LIN {X 0,Y 73.676,Z 293.865,A -85,B 0,C 180,E1 -30414.523,E2 -30414.523} C_VEL
LIN {X 0,Y 74.432,Z 292.814,A -85,B 0,C 180,E1 -30419.997,E2 -30419.997} C_VEL
LIN {X 0,Y 73.431,Z 293.677,A -85,B 0,C 180,E1 -30426.603,E2 -30426.603} C_VEL
LIN {X 0,Y 72.907,Z 294.465,A -85,B 0,C 180,E1 -30431.113,E2 -30431.113} C_VEL
LIN {X 0,Y 72.2,Z 295.883,A -85,B 0,C 180,E1 -30436.976,E2 -30436.976} C_VEL
LIN {X 0,Y 70.658,Z 298.436,A -85,B 0,C 180,E1 -30443.441,E2 -30443.441} C_VEL
LIN {X 0,Y 69.644,Z 299.949,A -85,B 0,C 180,E1 -30447.198,E2 -30447.198} C_VEL
LIN {X 0,Y 67.365,Z 302.892,A -85,B 0,C 180,E1 -30453.425,E2 -30453.425} C_VEL
LIN {X 0,Y 63.424,Z 307.476,A -85,B 0,C 180,E1 -30464.197,E2 -30464.197} C_VEL
LIN {X 0,Y 61.844,Z 310.777,A -85,B 0,C 180,E1 -30475.376,E2 -30475.376} C_VEL
LIN {X 0,Y 62.437,Z 312.643,A -85,B 0,C 180,E1 -30484.215,E2 -30484.215} C_VEL
LIN {X 0,Y 67.085,Z 314.547,A -85,B 0,C 180,E1 -30497.906,E2 -30497.906} C_VEL
LIN {X 0,Y 71.285,Z 314.971,A -85,B 0,C 180,E1 -30504.342,E2 -30504.342} C_VEL
LIN {X 0,Y 76.406,Z 314.961,A -85,B 0,C 180,E1 -30510,E2 -30510} C_VEL
LIN {X 0,Y 70.707,Z 314.927,A -85,B 0,C 180,E1 -30516.332,E2 -30516.332} C_VEL
LIN {X 0,Y 65.554,Z 314.211,A -85,B 0,C 180,E1 -30525.243,E2 -30525.243} C_VEL
LIN {X 0,Y 62.272,Z 312.421,A -85,B 0,C 180,E1 -30536.836,E2 -30536.836} C_VEL
LIN {X 0,Y 61.936,Z 310.037,A -85,B 0,C 180,E1 -30547.417,E2 -30547.417} C_VEL
LIN {X 0,Y 64.396,Z 306.165,A -85,B 0,C 180,E1 -30559.098,E2 -30559.098} C_VEL
LIN {X 0,Y 67.359,Z 302.893,A -85,B 0,C 180,E1 -30566.583,E2 -30566.583} C_VEL
LIN {X 0,Y 69.605,Z 299.971,A -85,B 0,C 180,E1 -30572.791,E2 -30572.791} C_VEL
LIN {X 0,Y 71.492,Z 297.039,A -85,B 0,C 180,E1 -30579.878,E2 -30579.878} C_VEL
LIN {X 0,Y 72.19,Z 295.89,A -85,B 0,C 180,E1 -30583.022,E2 -30583.022} C_VEL
LIN {X 0,Y 72.906,Z 294.466,A -85,B 0,C 180,E1 -30588.887,E2 -30588.887} C_VEL
LIN {X 0,Y 73.634,Z 293.478,A -85,B 0,C 180,E1 -30594.526,E2 -30594.526} C_VEL
LIN {X 0,Y 74.44,Z 292.808,A -85,B 0,C 180,E1 -30600.003,E2 -30600.003} C_VEL
LIN {X 0,Y 73.487,Z 294.094,A -85,B 0,C 180,E1 -30606.279,E2 -30606.279} C_VEL
LIN {X 0,Y 72.295,Z 295.22,A -85,B 0,C 180,E1 -30608.406,E2 -30608.406} C_VEL
LIN {X 0,Y 69.831,Z 297.145,A -85,B 0,C 180,E1 -30610.311,E2 -30610.311} C_VEL
LIN {X 0,Y 67.327,Z 298.912,A -85,B 0,C 180,E1 -30611.434,E2 -30611.434} C_VEL
LIN {X 0,Y 57.475,Z 304.685,A -85,B 0,C 180,E1 -30614.417,E2 -30614.417} C_VEL
LIN {X 0,Y 48.227,Z 309.171,A -85,B 0,C 180,E1 -30618.7,E2 -30618.7} C_VEL
LIN {X 0,Y 38.879,Z 312.786,A -85,B 0,C 180,E1 -30625.335,E2 -30625.335} C_VEL
LIN {X 0,Y 33.035,Z 314.591,A -85,B 0,C 180,E1 -30631.685,E2 -30631.685} C_VEL
LIN {X 0,Y 23.562,Z 317.062,A -85,B 0,C 180,E1 -30653.377,E2 -30653.377} C_VEL
LIN {X 0,Y 20.768,Z 317.664,A -85,B 0,C 180,E1 -30670.221,E2 -30670.221} C_VEL
LIN {X 0,Y 20.025,Z 317.831,A -85,B 0,C 180,E1 -30690,E2 -30690} C_VEL
LIN {X 0,Y 20.768,Z 317.664,A -85,B 0,C 180,E1 -30709.779,E2 -30709.779} C_VEL
LIN {X 0,Y 23.562,Z 317.062,A -85,B 0,C 180,E1 -30726.623,E2 -30726.623} C_VEL
LIN {X 0,Y 33.035,Z 314.591,A -85,B 0,C 180,E1 -30748.315,E2 -30748.315} C_VEL
LIN {X 0,Y 41.94,Z 311.634,A -85,B 0,C 180,E1 -30757.168,E2 -30757.168} C_VEL
LIN {X 0,Y 51.467,Z 307.64,A -85,B 0,C 180,E1 -30762.914,E2 -30762.914} C_VEL
LIN {X 0,Y 61.31,Z 302.505,A -85,B 0,C 180,E1 -30766.98,E2 -30766.98} C_VEL
LIN {X 0,Y 64.639,Z 300.584,A -85,B 0,C 180,E1 -30768.106,E2 -30768.106} C_VEL
LIN {X 0,Y 66.852,Z 298.764,A -85,B 0,C 180,E1 -30771.244,E2 -30771.244} C_VEL
LIN {X 0,Y 67.395,Z 298.046,A -85,B 0,C 180,E1 -30774.011,E2 -30774.011} C_VEL
LIN {X 0,Y 68.442,Z 296.911,A -85,B 0,C 180,E1 -30779.997,E2 -30779.997} C_VEL
LIN {X 0,Y 67.508,Z 297.553,A -85,B 0,C 180,E1 -30785.972,E2 -30785.972} C_VEL
LIN {X 0,Y 66.682,Z 298.624,A -85,B 0,C 180,E1 -30792.165,E2 -30792.165} C_VEL
LIN {X 0,Y 65.976,Z 299.629,A -85,B 0,C 180,E1 -30796.524,E2 -30796.524} C_VEL
LIN {X 0,Y 64.231,Z 301.578,A -85,B 0,C 180,E1 -30802.513,E2 -30802.513} C_VEL
LIN {X 0,Y 62.878,Z 303.159,A -85,B 0,C 180,E1 -30806.6,E2 -30806.6} C_VEL
LIN {X 0,Y 61.26,Z 304.717,A -85,B 0,C 180,E1 -30810.636,E2 -30810.636} C_VEL
LIN {X 0,Y 58.689,Z 307.105,A -85,B 0,C 180,E1 -30816.776,E2 -30816.776} C_VEL
LIN {X 0,Y 55.19,Z 311.025,A -85,B 0,C 180,E1 -30830.454,E2 -30830.454} C_VEL
LIN {X 0,Y 55.208,Z 313.32,A -85,B 0,C 180,E1 -30843.003,E2 -30843.003} C_VEL
LIN {X 0,Y 58.568,Z 314.807,A -85,B 0,C 180,E1 -30856.114,E2 -30856.114} C_VEL
LIN {X 0,Y 63.482,Z 315.319,A -85,B 0,C 180,E1 -30865.075,E2 -30865.075} C_VEL
LIN {X 0,Y 67.402,Z 315.229,A -85,B 0,C 180,E1 -30870,E2 -30870} C_VEL
LIN {X 0,Y 62.433,Z 315.236,A -85,B 0,C 180,E1 -30876.463,E2 -30876.463} C_VEL
LIN {X 0,Y 58.179,Z 314.746,A -85,B 0,C 180,E1 -30884.909,E2 -30884.909} C_VEL
LIN {X 0,Y 54.905,Z 312.671,A -85,B 0,C 180,E1 -30900.797,E2 -30900.797} C_VEL
LIN {X 0,Y 55.809,Z 309.953,A -85,B 0,C 180,E1 -30913.831,E2 -30913.831} C_VEL
LIN {X 0,Y 59.644,Z 306.186,A -85,B 0,C 180,E1 -30925.57,E2 -30925.57} C_VEL
LIN {X 0,Y 61.252,Z 304.718,A -85,B 0,C 180,E1 -30929.376,E2 -30929.376} C_VEL
LIN {X 0,Y 62.893,Z 303.139,A -85,B 0,C 180,E1 -30933.454,E2 -30933.454} C_VEL
LIN {X 0,Y 64.239,Z 301.573,A -85,B 0,C 180,E1 -30937.489,E2 -30937.489} C_VEL
LIN {X 0,Y 65.956,Z 299.631,A -85,B 0,C 180,E1 -30943.534,E2 -30943.534} C_VEL
LIN {X 0,Y 66.682,Z 298.625,A -85,B 0,C 180,E1 -30947.835,E2 -30947.835} C_VEL
LIN {X 0,Y 67.507,Z 297.554,A -85,B 0,C 180,E1 -30954.028,E2 -30954.028} C_VEL
LIN {X 0,Y 68.451,Z 296.906,A -85,B 0,C 180,E1 -30960.003,E2 -30960.003} C_VEL
LIN {X 0,Y 67.396,Z 298.046,A -85,B 0,C 180,E1 -30965.989,E2 -30965.989} C_VEL
LIN {X 0,Y 66.842,Z 298.771,A -85,B 0,C 180,E1 -30968.756,E2 -30968.756} C_VEL
LIN {X 0,Y 64.638,Z 300.584,A -85,B 0,C 180,E1 -30971.891,E2 -30971.891} C_VEL
LIN {X 0,Y 57.475,Z 304.685,A -85,B 0,C 180,E1 -30974.417,E2 -30974.417} C_VEL
LIN {X 0,Y 52.268,Z 307.16,A -85,B 0,C 180,E1 -30975.88,E2 -30975.88} C_VEL
LIN {X 0,Y 46.76,Z 309.424,A -85,B 0,C 180,E1 -30976.537,E2 -30976.537} C_VEL
LIN {X 0,Y 35.413,Z 312.966,A -85,B 0,C 180,E1 -30977.654,E2 -30977.654} C_VEL
LIN {X 0,Y 28.967,Z 314.652,A -85,B 0,C 180,E1 -30980.959,E2 -30980.959} C_VEL
LIN {X 0,Y 28.103,Z 314.782,A -85,B 0,C 180,E1 -30981.829,E2 -30981.829} C_VEL
LIN {X 0,Y 18.343,Z 316.85,A -85,B 0,C 180,E1 -30999.98,E2 -30999.98} C_VEL
LIN {X 0,Y 14.272,Z 317.452,A -85,B 0,C 180,E1 -31020.499,E2 -31020.499} C_VEL
LIN {X 0,Y 12.932,Z 317.619,A -85,B 0,C 180,E1 -31050,E2 -31050} C_VEL
LIN {X 0,Y 14.272,Z 317.452,A -85,B 0,C 180,E1 -31079.501,E2 -31079.501} C_VEL
LIN {X 0,Y 18.343,Z 316.85,A -85,B 0,C 180,E1 -31100.02,E2 -31100.02} C_VEL
LIN {X 0,Y 29.911,Z 314.379,A -85,B 0,C 180,E1 -31120.026,E2 -31120.026} C_VEL
LIN {X 0,Y 39.721,Z 311.422,A -85,B 0,C 180,E1 -31126.688,E2 -31126.688} C_VEL
LIN {X 0,Y 49.842,Z 307.428,A -85,B 0,C 180,E1 -31130.762,E2 -31130.762} C_VEL
LIN {X 0,Y 60.104,Z 302.292,A -85,B 0,C 180,E1 -31133.638,E2 -31133.638} C_VEL
LIN {X 0,Y 61.567,Z 301.26,A -85,B 0,C 180,E1 -31136.724,E2 -31136.724} C_VEL
LIN {X 0,Y 62.204,Z 300.755,A -85,B 0,C 180,E1 -31139.996,E2 -31139.996} C_VEL
LIN {X 0,Y 61.149,Z 301.337,A -85,B 0,C 180,E1 -31146.596,E2 -31146.596} C_VEL
LIN {X 0,Y 60.018,Z 302.426,A -85,B 0,C 180,E1 -31153.54,E2 -31153.54} C_VEL
LIN {X 0,Y 58.976,Z 303.467,A -85,B 0,C 180,E1 -31157.574,E2 -31157.574} C_VEL
LIN {X 0,Y 57.606,Z 304.623,A -85,B 0,C 180,E1 -31161.465,E2 -31161.465} C_VEL
LIN {X 0,Y 55.306,Z 306.438,A -85,B 0,C 180,E1 -31167.189,E2 -31167.189} C_VEL
LIN {X 0,Y 51.729,Z 309.05,A -85,B 0,C 180,E1 -31175.398,E2 -31175.398} C_VEL
LIN {X 0,Y 48.707,Z 311.604,A -85,B 0,C 180,E1 -31186.169,E2 -31186.169} C_VEL
LIN {X 0,Y 48.237,Z 314.159,A -85,B 0,C 180,E1 -31204.082,E2 -31204.082} C_VEL
LIN {X 0,Y 50.802,Z 315.149,A -85,B 0,C 180,E1 -31215.539,E2 -31215.539} C_VEL
LIN {X 0,Y 56.301,Z 315.561,A -85,B 0,C 180,E1 -31226.933,E2 -31226.933} C_VEL
LIN {X 0,Y 58.456,Z 315.495,A -85,B 0,C 180,E1 -31230,E2 -31230} C_VEL
LIN {X 0,Y 53.713,Z 315.497,A -85,B 0,C 180,E1 -31237.518,E2 -31237.518} C_VEL
LIN {X 0,Y 50.266,Z 315.063,A -85,B 0,C 180,E1 -31246.238,E2 -31246.238} C_VEL
LIN {X 0,Y 48.014,Z 313.88,A -85,B 0,C 180,E1 -31258.579,E2 -31258.579} C_VEL
LIN {X 0,Y 49.072,Z 311.272,A -85,B 0,C 180,E1 -31275.732,E2 -31275.732} C_VEL
LIN {X 0,Y 53.182,Z 308.076,A -85,B 0,C 180,E1 -31288.094,E2 -31288.094} C_VEL
LIN {X 0,Y 55.302,Z 306.438,A -85,B 0,C 180,E1 -31292.82,E2 -31292.82} C_VEL
LIN {X 0,Y 57.608,Z 304.622,A -85,B 0,C 180,E1 -31298.536,E2 -31298.536} C_VEL
LIN {X 0,Y 58.962,Z 303.468,A -85,B 0,C 180,E1 -31302.468,E2 -31302.468} C_VEL
LIN {X 0,Y 60.004,Z 302.434,A -85,B 0,C 180,E1 -31306.456,E2 -31306.456} C_VEL
LIN {X 0,Y 61.148,Z 301.338,A -85,B 0,C 180,E1 -31313.404,E2 -31313.404} C_VEL
LIN {X 0,Y 62.211,Z 300.752,A -85,B 0,C 180,E1 -31320.004,E2 -31320.004} C_VEL
LIN {X 0,Y 61.569,Z 301.259,A -85,B 0,C 180,E1 -31323.275,E2 -31323.275} C_VEL
LIN {X 0,Y 60.103,Z 302.292,A -85,B 0,C 180,E1 -31326.359,E2 -31326.359} C_VEL
LIN {X 0,Y 49.841,Z 307.428,A -85,B 0,C 180,E1 -31329.232,E2 -31329.232} C_VEL
LIN {X 0,Y 39.721,Z 311.422,A -85,B 0,C 180,E1 -31333.311,E2 -31333.311} C_VEL
LIN {X 0,Y 29.911,Z 314.379,A -85,B 0,C 180,E1 -31339.973,E2 -31339.973} C_VEL
LIN {X 0,Y 28.103,Z 314.782,A -85,B 0,C 180,E1 -31341.829,E2 -31341.829} C_VEL
LIN {X 0,Y 22.824,Z 315.916,A -85,B 0,C 180,E1 -31347.349,E2 -31347.349} C_VEL
LIN {X 0,Y 17.343,Z 316.751,A -85,B 0,C 180,E1 -31353.544,E2 -31353.544} C_VEL
LIN {X 0,Y 7.303,Z 317.435,A -85,B 0,C 180,E1 -31387.187,E2 -31387.187} C_VEL
LIN {X 0,Y 7.44,Z 317.287,A -85,B 0,C 180,E1 -31452.841,E2 -31452.841} C_VEL
LIN {X 0,Y 14.811,Z 316.638,A -85,B 0,C 180,E1 -31481.619,E2 -31481.619} C_VEL
LIN {X 0,Y 28.281,Z 314.167,A -85,B 0,C 180,E1 -31493.729,E2 -31493.729} C_VEL
LIN {X 0,Y 38.706,Z 311.21,A -85,B 0,C 180,E1 -31497.009,E2 -31497.009} C_VEL
LIN {X 0,Y 49.203,Z 307.215,A -85,B 0,C 180,E1 -31499.006,E2 -31499.006} C_VEL
LIN {X 0,Y 55.771,Z 304.239,A -85,B 0,C 180,E1 -31499.996,E2 -31499.996} C_VEL
LIN {X 0,Y 54.505,Z 304.848,A -85,B 0,C 180,E1 -31507.404,E2 -31507.404} C_VEL
LIN {X 0,Y 52.596,Z 306.118,A -85,B 0,C 180,E1 -31515.496,E2 -31515.496} C_VEL
LIN {X 0,Y 51.7,Z 306.717,A -85,B 0,C 180,E1 -31517.909,E2 -31517.909} C_VEL
LIN {X 0,Y 49.646,Z 308.09,A -85,B 0,C 180,E1 -31522.669,E2 -31522.669} C_VEL
LIN {X 0,Y 45.47,Z 310.437,A -85,B 0,C 180,E1 -31531.779,E2 -31531.779} C_VEL
LIN {X 0,Y 41.435,Z 313.169,A -85,B 0,C 180,E1 -31547.278,E2 -31547.278} C_VEL
LIN {X 0,Y 42.112,Z 315.318,A -85,B 0,C 180,E1 -31570.502,E2 -31570.502} C_VEL
LIN {X 0,Y 45.091,Z 315.757,A -85,B 0,C 180,E1 -31581.033,E2 -31581.033} C_VEL
LIN {X 0,Y 49.61,Z 315.758,A -85,B 0,C 180,E1 -31590,E2 -31590} C_VEL
LIN {X 0,Y 43.44,Z 315.544,A -85,B 0,C 180,E1 -31603.919,E2 -31603.919} C_VEL
LIN {X 0,Y 40.846,Z 314.409,A -85,B 0,C 180,E1 -31621.076,E2 -31621.076} C_VEL
LIN {X 0,Y 42.402,Z 312.317,A -85,B 0,C 180,E1 -31638.479,E2 -31638.479} C_VEL
LIN {X 0,Y 48.023,Z 308.977,A -85,B 0,C 180,E1 -31653.962,E2 -31653.962} C_VEL
LIN {X 0,Y 49.636,Z 308.095,A -85,B 0,C 180,E1 -31657.32,E2 -31657.32} C_VEL
LIN {X 0,Y 51.695,Z 306.717,A -85,B 0,C 180,E1 -31662.11,E2 -31662.11} C_VEL
LIN {X 0,Y 52.574,Z 306.128,A -85,B 0,C 180,E1 -31664.497,E2 -31664.497} C_VEL
LIN {X 0,Y 54.481,Z 304.859,A -85,B 0,C 180,E1 -31672.592,E2 -31672.592} C_VEL
LIN {X 0,Y 55.769,Z 304.24,A -85,B 0,C 180,E1 -31680.004,E2 -31680.004} C_VEL
LIN {X 0,Y 45.698,Z 308.747,A -85,B 0,C 180,E1 -31681.54,E2 -31681.54} C_VEL
LIN {X 0,Y 35.221,Z 312.362,A -85,B 0,C 180,E1 -31683.89,E2 -31683.89} C_VEL
LIN {X 0,Y 25.513,Z 314.73,A -85,B 0,C 180,E1 -31687.675,E2 -31687.675} C_VEL
LIN {X 0,Y 14.811,Z 316.638,A -85,B 0,C 180,E1 -31698.381,E2 -31698.381} C_VEL
LIN {X 0,Y 8.809,Z 317.24,A -85,B 0,C 180,E1 -31717.08,E2 -31717.08} C_VEL
LIN {X 0,Y 5.826,Z 317.408,A -85,B 0,C 180,E1 -31770,E2 -31770} C_VEL
LIN {X 0,Y 7.44,Z 317.287,A -85,B 0,C 180,E1 -31812.841,E2 -31812.841} C_VEL
LIN {X 0,Y 10.157,Z 317.105,A -85,B 0,C 180,E1 -31831.608,E2 -31831.608} C_VEL
LIN {X 0,Y 16.471,Z 316.308,A -85,B 0,C 180,E1 -31852.457,E2 -31852.457} C_VEL
LIN {X 0,Y 27.155,Z 314.271,A -85,B 0,C 180,E1 -31865.805,E2 -31865.805} C_VEL
LIN {X 0,Y 32.844,Z 312.828,A -85,B 0,C 180,E1 -31867.673,E2 -31867.673} C_VEL
LIN {X 0,Y 34.762,Z 312.328,A -85,B 0,C 180,E1 -31867.704,E2 -31867.704} C_VEL
LIN {X 0,Y 42.531,Z 309.777,A -85,B 0,C 180,E1 -31867.493,E2 -31867.493} C_VEL
LIN {X 0,Y 47.29,Z 308.048,A -85,B 0,C 180,E1 -31868.542,E2 -31868.542} C_VEL
LIN {X 0,Y 44.164,Z 309.551,A -85,B 0,C 180,E1 -31877.296,E2 -31877.296} C_VEL
LIN {X 0,Y 39.45,Z 311.758,A -85,B 0,C 180,E1 -31887.034,E2 -31887.034} C_VEL
LIN {X 0,Y 35.792,Z 313.416,A -85,B 0,C 180,E1 -31898.24,E2 -31898.24} C_VEL
LIN {X 0,Y 34.255,Z 315.569,A -85,B 0,C 180,E1 -31925.775,E2 -31925.775} C_VEL
LIN {X 0,Y 36.636,Z 316.012,A -85,B 0,C 180,E1 -31938.94,E2 -31938.94} C_VEL
LIN {X 0,Y 40.88,Z 316.018,A -85,B 0,C 180,E1 -31950,E2 -31950} C_VEL
LIN {X 0,Y 36.076,Z 315.941,A -85,B 0,C 180,E1 -31963.106,E2 -31963.106} C_VEL
LIN {X 0,Y 33.803,Z 314.999,A -85,B 0,C 180,E1 -31983.744,E2 -31983.744} C_VEL
LIN {X 0,Y 36.495,Z 313.022,A -85,B 0,C 180,E1 -32004.717,E2 -32004.717} C_VEL
LIN {X 0,Y 39.438,Z 311.758,A -85,B 0,C 180,E1 -32013.001,E2 -32013.001} C_VEL
LIN {X 0,Y 44.162,Z 309.551,A -85,B 0,C 180,E1 -32022.713,E2 -32022.713} C_VEL
LIN {X 0,Y 47.271,Z 308.057,A -85,B 0,C 180,E1 -32031.455,E2 -32031.455} C_VEL
LIN {X 0,Y 42.531,Z 309.777,A -85,B 0,C 180,E1 -32032.504,E2 -32032.504} C_VEL
LIN {X 0,Y 35.456,Z 312.15,A -85,B 0,C 180,E1 -32032.336,E2 -32032.336} C_VEL
LIN {X 0,Y 28.399,Z 313.955,A -85,B 0,C 180,E1 -32031.837,E2 -32031.837} C_VEL
LIN {X 0,Y 14.269,Z 316.426,A -85,B 0,C 180,E1 -32030.086,E2 -32030.086} C_VEL
LIN {X 0,Y 7.252,Z 317.029,A -85,B 0,C 180,E1 -32025.719,E2 -32025.719} C_VEL
LIN {X 0,Y 1.286,Z 317.196,A -85,B 0,C 180,E1 -31950,E2 -31950} C_VEL
LIN {X 0,Y 7.252,Z 317.029,A -85,B 0,C 180,E1 -31874.281,E2 -31874.281} C_VEL
LIN {X 0,Y 14.269,Z 316.426,A -85,B 0,C 180,E1 -31869.914,E2 -31869.914} C_VEL
LIN {X 0,Y 28.399,Z 313.955,A -85,B 0,C 180,E1 -31868.163,E2 -31868.163} C_VEL
LIN {X 0,Y 34.762,Z 312.328,A -85,B 0,C 180,E1 -31867.704,E2 -31867.704} C_VEL
LIN {X 0,Y 35.37,Z 312.181,A -85,B 0,C 180,E1 -31868.762,E2 -31868.762} C_VEL
LIN {X 0,Y 35.31,Z 312.238,A -85,B 0,C 180,E1 -31871.959,E2 -31871.959} C_VEL
LIN {X 0,Y 34.059,Z 312.666,A -85,B 0,C 180,E1 -31877.24,E2 -31877.24} C_VEL
LIN {X 0,Y 29.854,Z 314.217,A -85,B 0,C 180,E1 -31890.806,E2 -31890.806} C_VEL
LIN {X 0,Y 27.387,Z 315.165,A -85,B 0,C 180,E1 -31905.081,E2 -31905.081} C_VEL
LIN {X 0,Y 28.303,Z 316.266,A -85,B 0,C 180,E1 -31935.622,E2 -31935.622} C_VEL
LIN {X 0,Y 32.244,Z 316.275,A -85,B 0,C 180,E1 -31950,E2 -31950} C_VEL
LIN {X 0,Y 28.296,Z 316.267,A -85,B 0,C 180,E1 -31964.381,E2 -31964.381} C_VEL
LIN {X 0,Y 26.866,Z 315.563,A -85,B 0,C 180,E1 -31988.313,E2 -31988.313} C_VEL
LIN {X 0,Y 32.93,Z 313.109,A -85,B 0,C 180,E1 -32017.619,E2 -32017.619} C_VEL
LIN {X 0,Y 30.241,Z 313.743,A -85,B 0,C 180,E1 -32018.368,E2 -32018.368} C_VEL
LIN {X 0,Y 17.022,Z 316.213,A -85,B 0,C 180,E1 -32005.662,E2 -32005.662} C_VEL
LIN {X 0,Y 11.352,Z 316.817,A -85,B 0,C 180,E1 -31988.249,E2 -31988.249} C_VEL
LIN {X 0,Y 8.384,Z 316.985,A -85,B 0,C 180,E1 -31950,E2 -31950} C_VEL
LIN {X 0,Y 11.352,Z 316.817,A -85,B 0,C 180,E1 -31911.751,E2 -31911.751} C_VEL
LIN {X 0,Y 17.022,Z 316.213,A -85,B 0,C 180,E1 -31894.338,E2 -31894.338} C_VEL
LIN {X 0,Y 30.241,Z 313.743,A -85,B 0,C 180,E1 -31881.632,E2 -31881.632} C_VEL
LIN {X 0,Y 32.958,Z 313.103,A -85,B 0,C 180,E1 -31882.394,E2 -31882.394} C_VEL
LIN {X 0,Y 27.387,Z 315.165,A -85,B 0,C 180,E1 -31905.081,E2 -31905.081} C_VEL
LIN {X 0,Y 26.039,Z 315.585,A -85,B 0,C 180,E1 -31909.889,E2 -31909.889} C_VEL
LIN {X 0,Y 20.538,Z 316.352,A -85,B 0,C 180,E1 -31922.744,E2 -31922.744} C_VEL
LIN {X 0,Y 20.157,Z 316.506,A -85,B 0,C 180,E1 -31928.984,E2 -31928.984} C_VEL
LIN {X 0,Y 23.616,Z 316.532,A -85,B 0,C 180,E1 -31950,E2 -31950} C_VEL
LIN {X 0,Y 19.775,Z 316.378,A -85,B 0,C 180,E1 -31977.856,E2 -31977.856} C_VEL
LIN {X 0,Y 17.505,Z 316.605,A -85,B 0,C 180,E1 -31973.671,E2 -31973.671} C_VEL
LIN {X 0,Y 15.474,Z 316.774,A -85,B 0,C 180,E1 -31950,E2 -31950} C_VEL
LIN {X 0,Y 17.505,Z 316.605,A -85,B 0,C 180,E1 -31926.329,E2 -31926.329} C_VEL
LIN {X 0,Y 19.788,Z 316.377,A -85,B 0,C 180,E1 -31922.111,E2 -31922.111} C_VEL
LIN {X 0,Y 20.157,Z 316.506,A -85,B 0,C 180,E1 -31928.984,E2 -31928.984} C_VEL
LIN {X 0,Y 20.639,Z 318.503,A -85,B 0,C 180,E1 -31934.13,E2 -31934.13} C_VEL
LIN {X 0,Y 20.639,Z 600,A -85,B 0,C 180,E1 -31934.13,E2 -31934.13} C_VEL
LIN {X 0,Y 20.639,Z 600,A -85,B 0,C 180,E1 -31934.13,E2 -31934.13}

QRS_NEXT_CUT()

QRS_NEXT()
QRS_HOME()

END
